// Implicitly generated code : DO NOT EDIT
FUNCTION CheckLRangeSigned : LINT
VAR_INPUT
	value, lower, upper: LINT;
END_VAR

// Implicitly generated code : Only an Implementation suggestion
{noflow}
IF (value < lower) THEN
	CheckLRangeSigned := lower;
	G_Diag.uiCheckRange:=G_Diag.uiCheckRange+1;
ELSIF(value > upper) THEN
	CheckLRangeSigned := upper;
	G_Diag.uiCheckRange:=G_Diag.uiCheckRange+1;
ELSE
	CheckLRangeSigned := value;
END_IF

{flow}

END_FUNCTION

(* stored: Version 1.1.0.1, ProductVersion 3.1.4024.4
   POU CheckLRangeSigned: Id {58d556c4-89e7-415d-a773-dc7f22bfb992}, SpecialFunc CheckLRangeSigned *)
